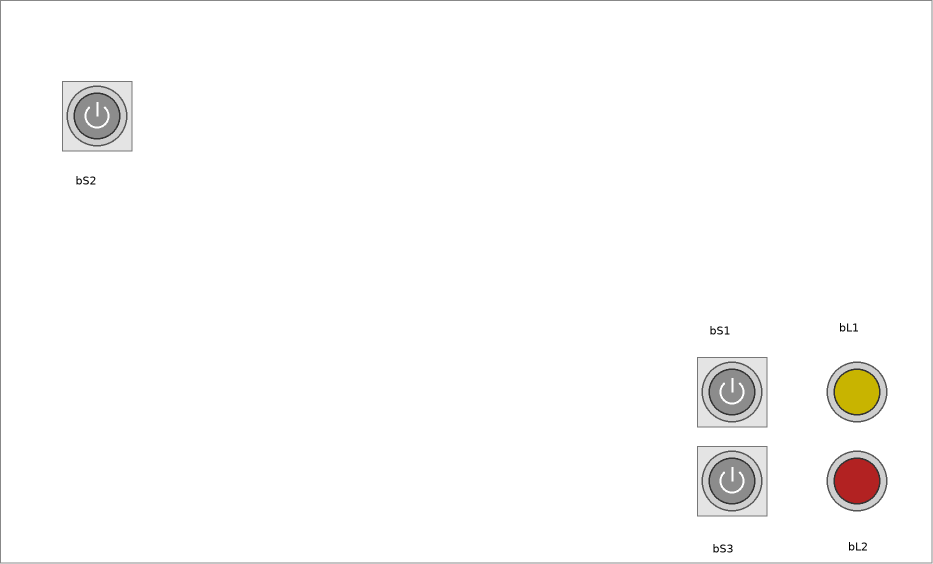
VISUALIZATION Visu  // 933x564
    Lamp1 (822,357 70x70), variable: MAIN.bL1, style: Lamp-Lamp1-Yellow
    PowerSwitch (697,357 70x70), variable: MAIN.bS1, behaviour: TAP, style: Switch-PowerSwitch-Gray
    Lamp1 (822,446 70x70), variable: MAIN.bL2, style: Lamp-Lamp1-Red
    PowerSwitch (697,446 70x70), variable: MAIN.bS3, behaviour: TAP, style: Switch-PowerSwitch-Gray
    Label (783,532 150x30), "bL2"
    Label (648,534 150x30), "bS3"
    Label (645,316 150x30), "bS1"
    Label (774,313 150x30), "bL1"
    PowerSwitch (62,81 70x70), variable: MAIN.bS2, behaviour: TAP, style: Switch-PowerSwitch-Gray
    Label (11,166 150x30), "bS2"
END_VISUALIZATION

(* stored: Version 1.1.0.1, ProductVersion 3.1.4024.12
   Visu Visu: Id {81112a8d-b048-418e-b6bf-51e471bbf6d5} *)
